Staubli VAL3: IO.pjx

--- IO.pjx ---
Parameters version=s7.8.3 stackSize=5000 millimeterUnit=true
Program file=CloseAll.pgx
Program file=getIO.pgx
Program file=Main.pgx
Program file=MainKey.pgx
Program file=OnF1.pgx
Program file=OnF2.pgx
Program file=OnF7.pgx
Program file=OnF8.pgx
Program file=Refresh.pgx
Program file=RefreshList.pgx
Program file=setIO.pgx
Program file=start.pgx
Program file=stop.pgx
Data file=IO.dtx
Library alias=user path=Disk://userPage/USERPAGE.pjx

--- IO.dtx ---
mdesc mNomSpeed
public dio diStart = {link=usrIn0}
public dio diStop
public dio diGanying
public dio diTab
public dio diXi
public dio dIn{}
  [dIn1] = {link=BasicIO-1\%I0}
  [dIn8] = {link=BasicIO-1\%I7}
  [dIn7] = {link=BasicIO-1\%I6}
  [dIn6] = {link=BasicIO-1\%I5}
  [dIn5] = {link=BasicIO-1\%I4}
  [dIn4] = {link=BasicIO-1\%I3}
  [dIn3] = {link=BasicIO-1\%I2}
  [dIn2] = {link=BasicIO-1\%I1}
  [dIn9] = {link=BasicIO-1\%I8}
  [dIn10] = {link=BasicIO-1\%I9}
  [dIn11] = {link=BasicIO-1\%I10}
  [dIn12] = {link=BasicIO-1\%I11}
  [dIn13] = {link=BasicIO-1\%I12}
  [dIn14] = {link=BasicIO-1\%I13}
  [dIn15] = {link=BasicIO-1\%I14}
  [dIn16] = {link=BasicIO-1\%I15}
public dio dOut{}
  [dOut1] = {link=BasicIO-1\%Q0}
  [dOut2] = {link=BasicIO-1\%Q1}
  [dOut3] = {link=BasicIO-1\%Q2}
  [dOut4] = {link=BasicIO-1\%Q3}
  [dOut5] = {link=BasicIO-1\%Q4}
  [dOut6] = {link=BasicIO-1\%Q5}
  [dOut7] = {link=BasicIO-1\%Q6}
  [dOut8] = {link=BasicIO-1\%Q7}
  [dOut9] = {link=BasicIO-1\%Q8}
  [dOut10] = {link=BasicIO-1\%Q9}
  [dOut11] = {link=BasicIO-1\%Q10}
  [dOut12] = {link=BasicIO-1\%Q11}
  [dOut13] = {link=BasicIO-1\%Q12}
  [dOut14] = {link=BasicIO-1\%Q13}
  [dOut15] = {link=BasicIO-1\%Q14}
  [dOut16] = {link=BasicIO-1\%Q15}
string sIOName
string sList
bool bListRefresh
bool bUserRefresh
bool bExit
num nType
num nSelected
string sItem
public dio diEndStop = {link=usrIn1}

--- Main.pgx ---
public program Main(num x_nType)
  local num l_nKey
begin
  //
  bUserRefresh=bListRefresh=true
  bExit=false
  nType=x_nType
  //
  do
    call Refresh()
    call RefreshList()
    call user:setList("工具",sList,bUserRefresh,bListRefresh,nSelected,sItem,l_nKey)
    bUserRefresh=false
    bListRefresh=false
    call MainKey(l_nKey)
    delay(0)
  until bExit

end

--- start.pgx ---
program start()
begin
  call Main(0)
end

--- CloseAll.pgx ---
public program CloseAll()
begin
  dOut["dOut1"]=false
  dOut["dOut2"]=false
  dOut["dOut3"]=false
  dOut["dOut4"]=false
  dOut["dOut5"]=false
  dOut["dOut6"]=false
  dOut["dOut7"]=false
  dOut["dOut8"]=false
  dOut["dOut9"]=false
  dOut["dOut10"]=false
  dOut["dOut11"]=false
  dOut["dOut12"]=false
  dOut["dOut13"]=false
  dOut["dOut14"]=false
  dOut["dOut15"]=false
  dOut["dOut16"]=false
end

--- getIO.pgx ---
public program getIO(string& x_sIO)
begin
  x_sIO=sIOName
end

--- OnF1.pgx ---
program OnF1()
begin
  //
  if nType==1
    call setIO(sItem)
    popUpMsg("选择IO："+sItem)
  endIf

end

--- OnF2.pgx ---
program OnF2()
begin
  //
  if find(sItem,"O")!=-1
    if dOut[sIOName]==true
      dOut[sIOName]=false
    endIf
  else
    popUpMsg("对输入量无效。")
  endIf


end

--- Refresh.pgx ---
program Refresh()
begin
  //
  if bUserRefresh
    cls()
    userPage()
    if nType==1
      gotoxy(1,1)
      put("F1->确定")
      gotoxy(1,13)
      put("F1")
    endIf

    gotoxy(1,2)
    put("F2->开/关")
    gotoxy(6,13)
    put("F2")
    //    gotoxy(1,3)
    //    put("F3->删除")
    //    gotoxy(11,13)
    //    put("F3")
    //    gotoxy(1,4)
    //    put("F4->编辑路径")
    //    gotoxy(16,13)
    //    put("编辑")
    //
    //    gotoxy(1,6)
    //    put("F6->")
    //    gotoxy(26,13)
    //    put("")
//    gotoxy(1,7)
//    put("F7->保存")
//    gotoxy(31,13)
//    put("F7")
    gotoxy(1,8)
    put("F8->返回")
    gotoxy(36,13)
    put("F8")
  endIf
end

--- RefreshList.pgx ---
program RefreshList()
  local num l_ni
begin
  //

  if bListRefresh
    resize(sList,1,32)
    for l_ni=0 to 15
      sList[l_ni]="dIn"+toString("",l_ni+1)
      sList[l_ni+15]="dOut"+toString("",l_ni+1)
    endFor
  endIf

end

--- setIO.pgx ---
public program setIO(string x_sIO)
begin
  //
  sIOName=x_sIO
end
